// TIA Portal V19 export
VAR_GLOBAL   // PLC tag table "D10"
   D10_Lp_EntryReq_LB201 AT %Q108.1 : Bool;   // 230SH1
   D10_Lp_SafetyReset_LB201 AT %Q108.2 : Bool;   // 230SH2
   D10_Pb_EntryReq_LB201 AT %I106.4 : Bool;   // 230SH1
   D10_Pb_SafetyReset_LB201 AT %I106.5 : Bool;   // 230SH2
   D10_Comando_Elettroserratura AT %Q108.0 : Bool;   // 23002
   D10_Cancello_Chiuso AT %I106.2 : Bool;   // 23001
   D10_Cancello_Bloccato AT %I106.3 : Bool;   // 23003
   D10_Ls_Os1 AT %I1072.1 : Bool;   // 105DI1 - 230A1
   D10_Ls_Os2 AT %I1072.5 : Bool;   // 105DI5 - 230A1
END_VAR
